RoboDK station: Tutorial_1.rdk

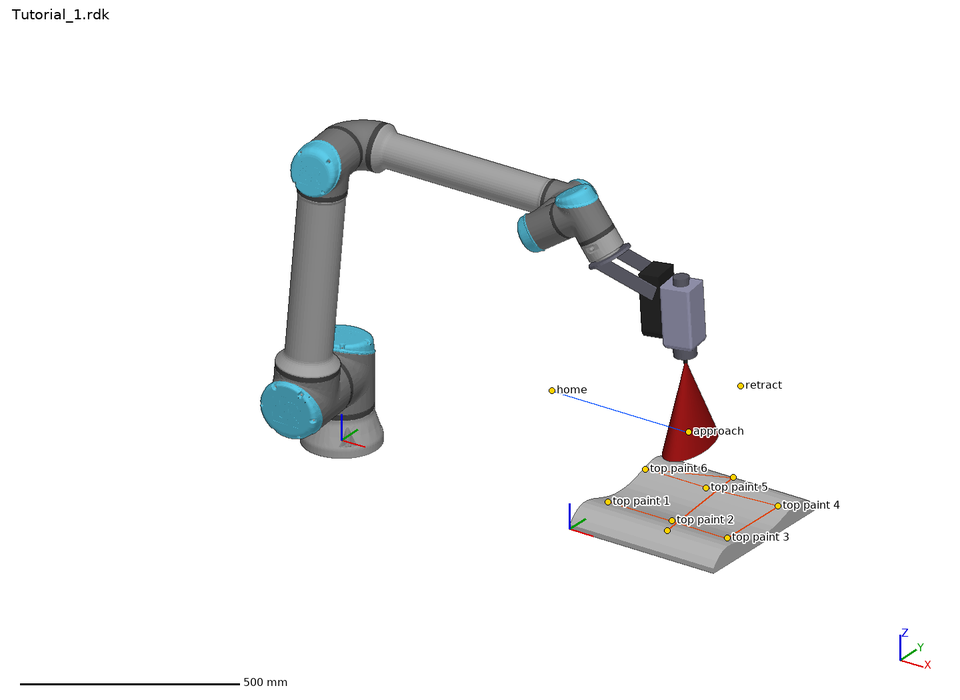
[picture v0: the station drawn from its stored meshes, robots at their saved joint values, targets as dots, program paths as lines]
Station Tutorial_1 (saved by RoboDK 5.7.4). Poses are relative to the parent item; angles as X-Y-Z fixed-axis rotations.
  - frame UR10e Base at (441.14, 132.2, 22.18) mm
    - robot UR10e: 6 axes, payload 10 kg, reach 1300 mm, repeatability 0.05 mm, weight 28.9 kg
        modified DH rows (alpha deg, a mm, theta deg, d mm): 0, 0, 0, 180.7; 90, 0, 180, 0; 0, 612.6, 0, 0; 0, 571.335, 0, 174.15; -90, 0, 0, 119.85; 90, 0, 180, 116.55
        joint limits [-360, -360, -360, -360, -360, -360] to [360, 360, 360, 360, 360, 360]; home [0, -90, -90, 0, 90, 0]; saved at [6.406, -94.812, -88.539, -53.391, 90.984, -271.554]
      - tool Paint gun, TCP at (50, 0, 450) mm, rotated rx 0 ry 30 rz 0 deg, size 203.2 x 279.7 x 471.5 mm
  - frame Frame 2 at (1245.62, -110.53, 118.17) mm
    - object Object Inspection at (0, 0, 0) mm, size 400 x 400 x 46.2 mm, geometry from Object Inspection.stp
    - target home (Cartesian target) at (257.42, -436.87, 597.72) mm, rotated rx 170.18 ry 60 rz 180 deg; joints [0, -90, -90, 10.87, 144.368, -264.599] of UR10e
    - target approach (Cartesian target) at (198.68, 188.54, 226.37) mm, rotated rx -179.97 ry 3.27 rz -171.75 deg; joints [6.406, -94.812, -88.539, -53.391, 90.984, -271.554] of UR10e
    - target top paint 1 (Cartesian target) at (35.38, 102.36, 37.97) mm, rotated rx -162.35 ry -2.09 rz -173.46 deg; joints [15.844, -101.263, -88.228, 126.026, -70.422, -90.419] of UR10e
    - target top paint 2 (Cartesian target) at (208.22, 109.56, 35.66) mm, rotated rx -162.35 ry -2.09 rz -173.46 deg; joints [12.767, -100.862, -100.291, -41.374, 71.82, -273.318] of UR10e
    - target top paint 3 (Cartesian target) at (363.35, 106.32, 36.7) mm, rotated rx -162.35 ry -2.09 rz -173.46 deg; joints [10.407, -115.006, -81.249, -45.609, 72.921, -275.507] of UR10e
    - target top paint 4 (Cartesian target) at (367.39, 303.39, 39.81) mm, rotated rx 162.31 ry 1.71 rz -174.67 deg; joints [3.401, -117, -80.433, -40.104, 106.302, -262.624] of UR10e
    - target top paint 5 (Cartesian target) at (173.58, 293.07, 36.5) mm, rotated rx 162.31 ry 1.71 rz -174.67 deg; joints [3.494, -100.033, -103.916, -33.565, 106.252, -262.542] of UR10e
    - target top paint 6 (Cartesian target) at (4.86, 292.72, 36.39) mm, rotated rx 162.31 ry 1.71 rz -174.67 deg; joints [4.511, -84.253, -120.447, -32.568, 105.704, -261.651] of UR10e
    - target top paint 7 (Cartesian target) at (190.04, 378.35, 32.94) mm, rotated rx -142.4 ry -1.94 rz -177.48 deg; joints [41.731, -109.868, -92.501, -64.767, 44.717, -243.014] of UR10e
    - target top paint 8 (Cartesian target) at (238.88, 47.15, 44.46) mm, rotated rx 168.49 ry 0.42 rz -177.96 deg; joints [-9.233, -108.419, -89.469, -43.412, 105.568, -274.214] of UR10e
    - target retract (Cartesian target) at (169.09, 437.78, 236.08) mm, rotated rx 178.43 ry 3.27 rz -171.75 deg; joints [25.284, -92.835, -89.559, -55.154, 82.066, -254.896] of UR10e
  - program ApproachMove (4 instructions, listed below)
  - program PaintTop (10 instructions, listed below)
  - program Retract (3 instructions, listed below)
  - program MainProgram (3 instructions, listed below)
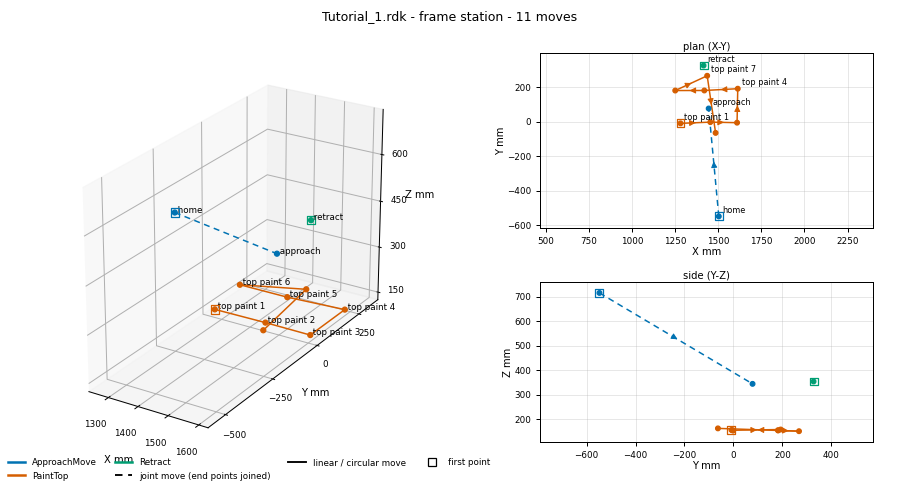
[picture p0: tool path of Tutorial_1.rdk in frame station, 11 of 11 moves have a stored position in this frame; points joined in program order, loops and branches not executed]

--- program ApproachMove (robot UR10e) ---
  Set Ref.: Frame 2
  Set Tool: Paint gun
  MoveJ (home)
  MoveJ (approach)

--- program PaintTop (robot UR10e) ---
  Set Ref.: Frame 2
  Set Tool: Paint gun
  MoveL (top paint 1)
  MoveL (top paint 2)
  MoveL (top paint 3)
  MoveL (top paint 4)
  MoveL (top paint 5)
  MoveL (top paint 6)
  MoveL (top paint 7)
  MoveL (top paint 8)

--- program Retract (robot UR10e) ---
  Set Ref.: Frame 2
  Set Tool: Paint gun
  MoveJ (retract)

--- program MainProgram (robot UR10e) ---
  Call ApproachMove
  Call PaintTop
  Call Retract
